// TIA Portal V17 export
// export: Created 2024-09-02T12:50:31.3063223Z, ExportSetting WithDefaults, DisplayName Totally Integrated Automation Portal, DisplayVersion V17, DisplayName TIA Portal Openness, DisplayVersion V17, DisplayName TIA Portal Version Control Interface, DisplayVersion V17, DisplayName STEP 7 Professional, DisplayVersion V17, DisplayName STEP 7 Safety, DisplayVersion V17, DisplayName WinCC Professional, DisplayVersion V17
TYPE "UFM_DataSample"
TITLE = UFM_DataSample
// Structure describing a measured value for the UFM5 library.
// stored: IsFailsafeCompliant false
   STRUCT
      New : Bool;   // New (vs. old)
      Ok : Bool;   // Ok (vs. NOk)
      Missed : Bool;   // Missed (vs. sampled)
      UpperLimitViolated : Bool;   // Upper limit violated
      LowerLimitViolated : Bool;   // Lower limit violated
      StartPosition : Real;   // Position (Start)
      EndPosition : Real;   // Position (End)
      UpperLimit : Real;   // Upper limit
      Value : Real;   // Force /Analog value
      LowerLimit : Real;   // Lower limit
      Position : Real;   // Position (when sampled)
   END_STRUCT;
END_TYPE
